# EPICS autosave request: iocBoot/sioc-esb-xps5/xpsm.req
$(P):MOTR:ABS1.VAL
$(P):MOTR:ABS2.VAL
$(P):MOTR:ABS3.VAL
$(P):MOTR:SAVED1.VAL
$(P):MOTR:SAVED2.VAL
$(P):MOTR:SAVED3.VAL
$(P):MOTR.HLM
$(P):MOTR.LLM
$(P):MOTR.DHLM
$(P):MOTR.DLLM
$(P):MOTR.SMAX
$(P):MOTR.S
$(P):MOTR.SBAK
$(P):MOTR.SBAS
$(P):MOTR.ACCL
$(P):MOTR.BACC
$(P):MOTR.BDST
$(P):MOTR.FRAC
$(P):MOTR.HVEL
$(P):MOTR.OFF
$(P):MOTR.EGU
$(P):MOTR.SREV
$(P):MOTR.UREV
$(P):MOTR.ERES
$(P):MOTR.RDBD
$(P):MOTR.PREC
$(P):MOTR.RTRY
$(P):MOTR.TWV
$(P):MOTR.RBV
